// return the norm of a vector
FUNCTION norm : LREAL
VAR_IN_OUT CONSTANT
	vec :ARRAY[*] OF LREAL;
END_VAR
VAR
	m,i:DINT;
END_VAR

m:=UPPER_BOUND(vec,1);
norm:=0;
FOR i:=1 TO m DO
	norm := norm + vec[i]*vec[i];
END_FOR

norm := SQRT(norm);

END_FUNCTION

(* stored: Version 1.1.0.1, ProductVersion 3.1.4024.12
   POU norm: Id {0015b5c6-4029-411f-8387-131591190194}, SpecialFunc None *)
